(* Logix 5000 project; controller DC01 vendor 1 type 14 code 165 rev 32.12; software revision 32.04; part 6 of 13 *)
(* tags used below, declared in another part *)
   Always_Off : BOOL;
   Barcode_Scan_ln02 : MESSAGE;
   Break_1stStation : BOOL;
   Break_LineWide : BOOL;
   Break_WorkCenter : BOOL;
   Break_Workstation : BOOL;
   FaultExists : CONTROL;
   LN02_MainLine_MSG : MESSAGE;
   Local_Timer : TIMER[30];
   local_timer2 : TIMER;
   ONS_0 : DINT;
   Scheduled_Units_Buffer : DINT;
   Shift_Reset : BOOL;
   Shift_Reset_ONS : BOOL;
   LN02_1st_Station_Break_Code : DINT;
   LN02_Additional_Break_Limit_Mins : DINT;
   LN02_Boxing_MNT : DINT;
   LN02_Ceran_MNT : DINT;
   LN02_Console_MNT : DINT;
   LN02_Cooktop_MNT : DINT;
   LN02_Current_Shift_Duration_Mins : DINT;
   LN02_Current_Shift_Duration_wBreaks_Mins : DINT;
   LN02_DC_Controlled_Theoretical_Units : BOOL;
   LN02_Door_MNT : DINT;
   LN02_FPY : REAL;
   LN02_FrontFrame_MNT : DINT;
   LN02_Ignition_NewSNModel : BOOL[32];
   LN02_Ignition_SNModelMSG : STRING[5];
   LN02_MachineOverAll_MNT : DINT;
   LN02_Main_Messages : DINT[250];
   LN02_MainBack_MNT : DINT;
   LN02_Messages_Barcode_SNModel : Barcode_SNModel;
   LN02_OT_Shift_Break_In_Minutes : DINT;
   LN02_OvenCavity_MNT : DINT;
   LN02_Schedule : UDT_Current_Status;
   LN02_Schedule_Cycle_Timer : TIMER;
   LN02_Schedule_Max_Break_Duration : DINT;
   LN02_Schedule_Max_Break_Timer : TIMER;
   LN02_Schedule_TAKT_REAL : REAL;
   LN02_SidePanels_MNT : DINT;
   LN02_Standard_Shift_Break_In_Minutes : DINT;
   LN02_StorageDrawer_MNT : DINT;
   LN02_Test_MNT : DINT;
   LN02_Theoretical_Units_Counter : COUNTER;
   LN02_Theoretical_Units_Counter_ONS : BOOL;
   LN02_Units_for_repair : DINT;
   LN02_Wiring_MNT : DINT;
   LN02ECM02 : DINT;
   LN02ECM03 : DINT;
   LN02ECM04 : DINT;
   LN02ECM05 : DINT;
   LN02EDM04 : DINT;
   LN02EDM06 : DINT;
   LN02EDM07 : DINT;
   LN02EEM01 : DINT;
   LN02EEM02 : DINT;
   LN02EHM01 : DINT;
   LN02EHM02 : DINT;
   LN02EHM03 : DINT;
   LN02EHM04 : DINT;
   LN02EHM05 : DINT;
   LN02EHM06 : DINT;
   LN02EHM07 : DINT;
   LN02EHM08 : DINT;
   LN02EHM09 : DINT;
   LN02EHM10 : DINT;
   LN02NAS03 : DINT;
   LN02NES01 : DINT;
   LN02NES02 : DINT;
   LN02NES03 : DINT;
   LN02NES04 : DINT;
   LN02NFS01 : DINT;
   LN02NFS02 : DINT;
   LN02SAS01 : DINT;
   LN02SAS02 : DINT;
   LN02SAS03 : DINT;
   LN02SBS01 : DINT;
   LN02SBS02 : DINT;
   LN02SBS03 : DINT;
   LN02SFS01 : DINT;
   LN02SFS02 : DINT;
   LN02SFS03 : DINT;
   LN02SFS04 : DINT;
   LN02WAM01 : DINT;
   LN02WBM01 : DINT;
   LN02WBM02 : DINT;
   LN02WBM03 : DINT;
   LN02WBM04 : DINT;
   LN02WCM01 : DINT;
   LN02WCM02 : DINT;
   LN02WCM03 : DINT;
   LN02WCM04 : DINT;
   LN02WCM05 : DINT;
   LN02WCM06 : DINT;
   LN02WDM01 : DINT;
   LN02WDM02 : DINT;
   LN02WDM03 : DINT;
   LN02WDM04 : DINT;
   LN02WDM05 : DINT;
   LN02WDM06 : DINT;
   LN02WEM01 : DINT;
   LN02WFM01 : DINT;
   LN02WGM01 : DINT;
   LN02WGS01 : DINT;
   LN02WGS02 : DINT;
   LN02WGS03 : DINT;
   LN02WGS04 : DINT;
(* LN02, continued *)

ROUTINE R02_CurrentShift_Calcs   (* ladder *)
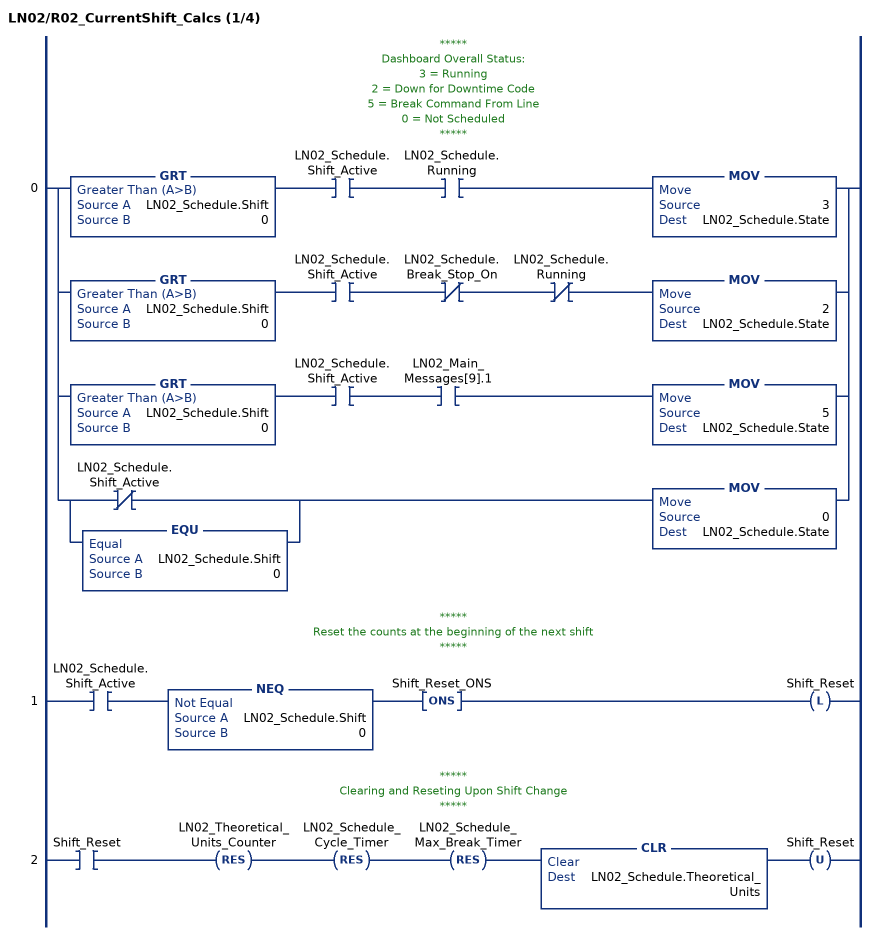
   // *****
   // Dashboard Overall Status:
   // 3 = Running
   // 2 = Down for Downtime Code
   // 5 = Break Command From Line
   // 0 = Not Scheduled
   // *****
   0: [GRT(LN02_Schedule.Shift,0) XIC(LN02_Schedule.Shift_Active) XIC(LN02_Schedule.Running) MOV(3,LN02_Schedule.State) ,GRT(LN02_Schedule.Shift,0) XIC(LN02_Schedule.Shift_Active) XIO(LN02_Schedule.Break_Stop_On) XIO(LN02_Schedule.Running) MOV(2,LN02_Schedule.State) ,GRT(LN02_Schedule.Shift,0) XIC(LN02_Schedule.Shift_Active) XIC(LN02_Main_Messages[9].1) MOV(5,LN02_Schedule.State) ,[XIO(LN02_Schedule.Shift_Active) ,EQU(LN02_Schedule.Shift,0) ] MOV(0,LN02_Schedule.State) ];
   // *****
   // Reset the counts at the beginning of the next shift
   // *****
   1: XIC(LN02_Schedule.Shift_Active)NEQ(LN02_Schedule.Shift,0)ONS(Shift_Reset_ONS)OTL(Shift_Reset);
   // *****
   // Clearing and Reseting Upon Shift Change
   // *****
   2: XIC(Shift_Reset)RES(LN02_Theoretical_Units_Counter)RES(LN02_Schedule_Cycle_Timer)RES(LN02_Schedule_Max_Break_Timer)CLR(LN02_Schedule.Theoretical_Units)OTU(Shift_Reset);
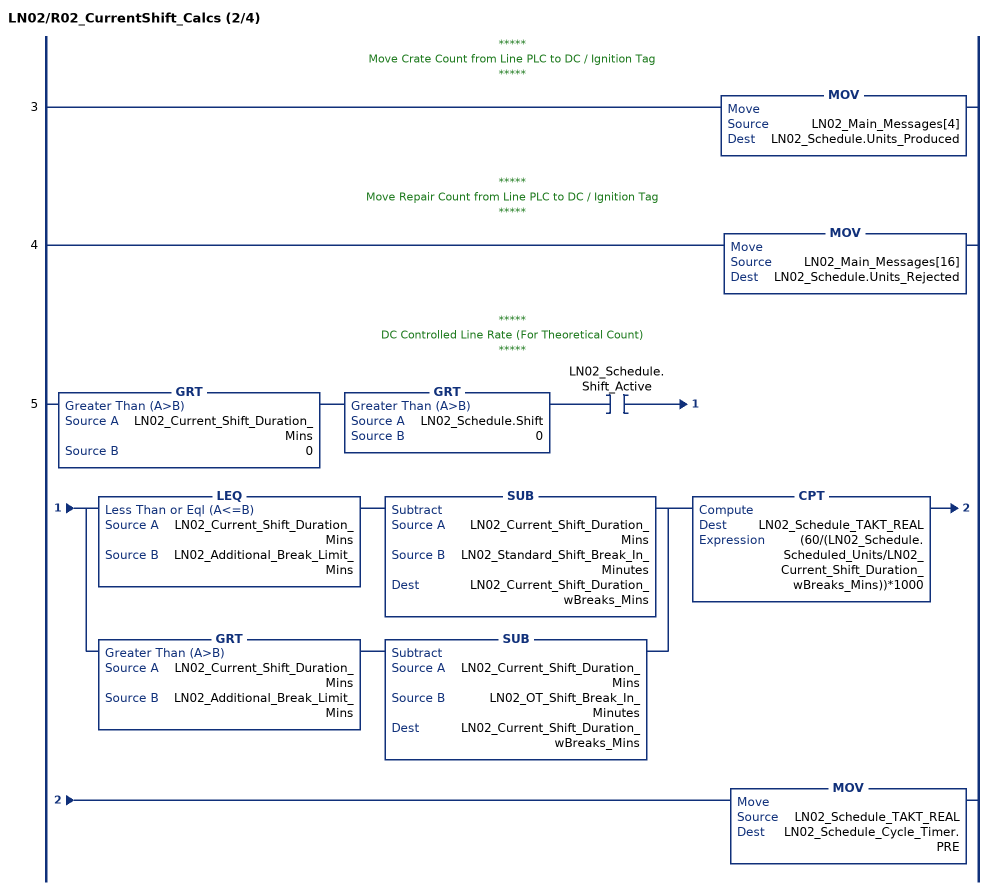
   // *****
   // Move Crate Count from Line PLC to DC / Ignition Tag
   // *****
   3: MOV(LN02_Main_Messages[4],LN02_Schedule.Units_Produced);
   // *****
   // Move Repair Count from Line PLC to DC / Ignition Tag
   // *****
   4: MOV(LN02_Main_Messages[16],LN02_Schedule.Units_Rejected);
   // *****
   // DC Controlled Line Rate (For Theoretical Count)
   // *****
   5: GRT(LN02_Current_Shift_Duration_Mins,0)GRT(LN02_Schedule.Shift,0)XIC(LN02_Schedule.Shift_Active)[LEQ(LN02_Current_Shift_Duration_Mins,LN02_Additional_Break_Limit_Mins) SUB(LN02_Current_Shift_Duration_Mins,LN02_Standard_Shift_Break_In_Minutes,LN02_Current_Shift_Duration_wBreaks_Mins) ,GRT(LN02_Current_Shift_Duration_Mins,LN02_Additional_Break_Limit_Mins) SUB(LN02_Current_Shift_Duration_Mins,LN02_OT_Shift_Break_In_Minutes,LN02_Current_Shift_Duration_wBreaks_Mins) ]CPT(LN02_Schedule_TAKT_REAL,(60/(LN02_Schedule.Scheduled_Units/LN02_Current_Shift_Duration_wBreaks_Mins))*1000)MOV(LN02_Schedule_TAKT_REAL,LN02_Schedule_Cycle_Timer.PRE);
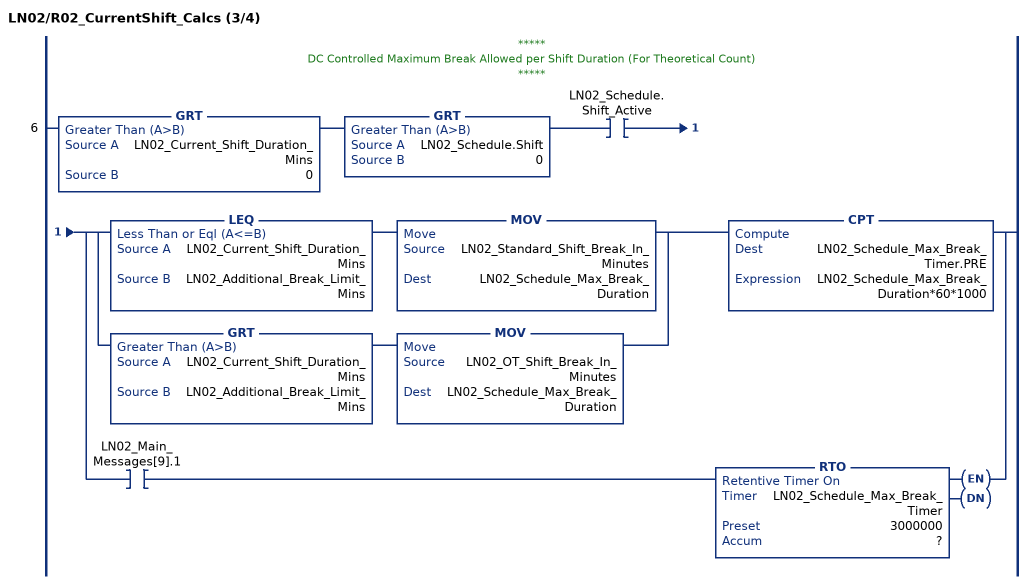
   // *****
   // DC Controlled Maximum Break Allowed per Shift Duration (For Theoretical Count)
   // *****
   6: GRT(LN02_Current_Shift_Duration_Mins,0)GRT(LN02_Schedule.Shift,0)XIC(LN02_Schedule.Shift_Active)[[LEQ(LN02_Current_Shift_Duration_Mins,LN02_Additional_Break_Limit_Mins) MOV(LN02_Standard_Shift_Break_In_Minutes,LN02_Schedule_Max_Break_Duration) ,GRT(LN02_Current_Shift_Duration_Mins,LN02_Additional_Break_Limit_Mins) MOV(LN02_OT_Shift_Break_In_Minutes,LN02_Schedule_Max_Break_Duration) ] CPT(LN02_Schedule_Max_Break_Timer.PRE,LN02_Schedule_Max_Break_Duration*60*1000) ,XIC(LN02_Main_Messages[9].1) RTO(LN02_Schedule_Max_Break_Timer,?,?) ];
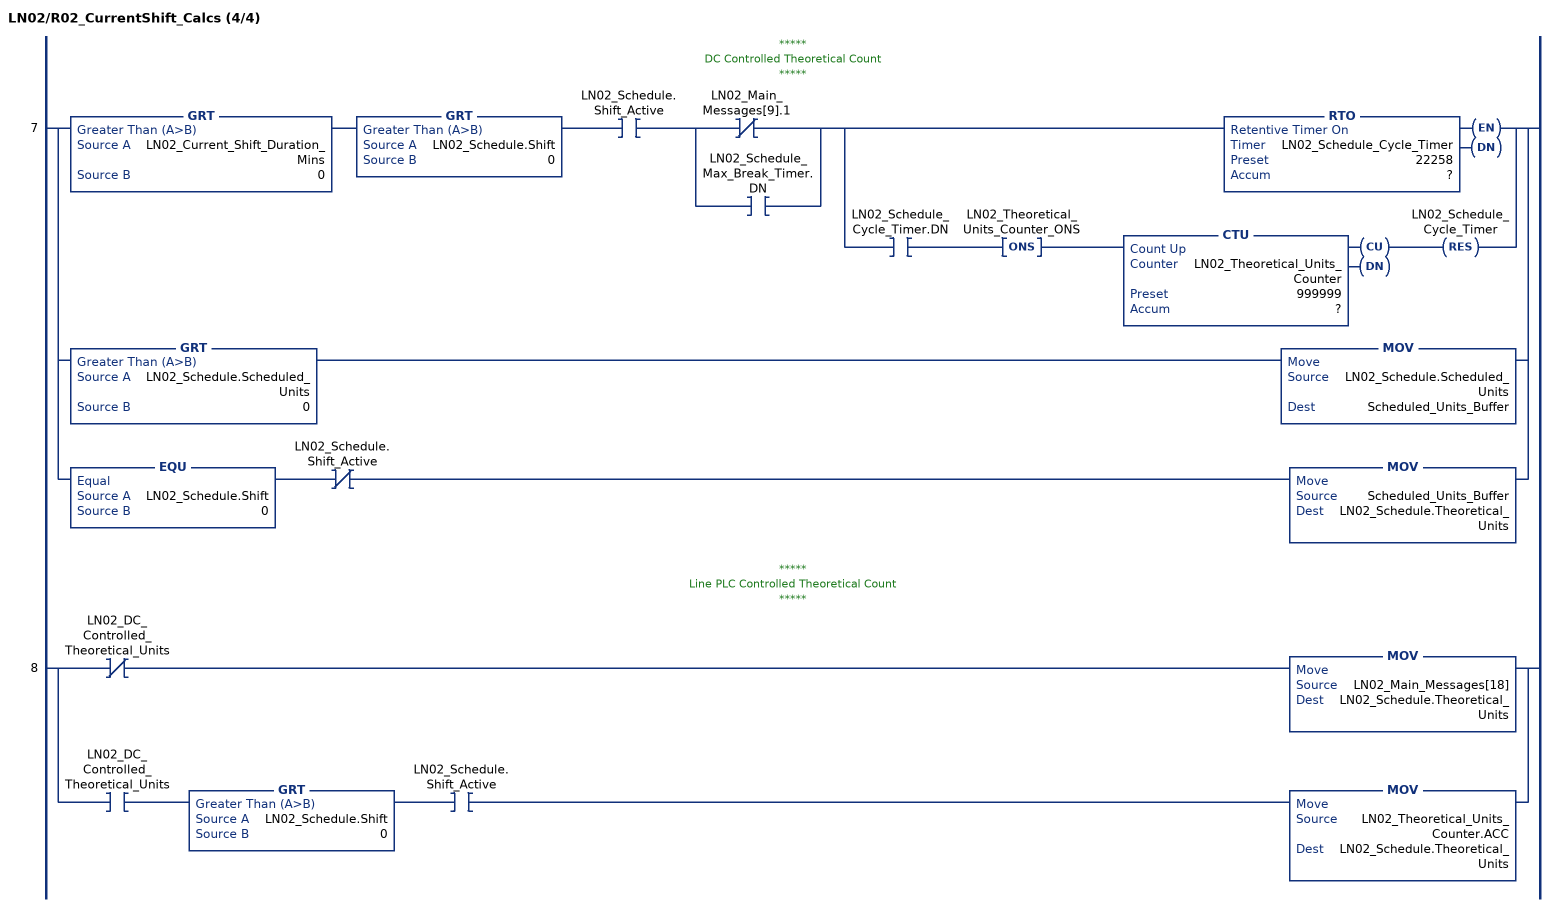
   // *****
   // DC Controlled Theoretical Count
   // *****
   7: [GRT(LN02_Current_Shift_Duration_Mins,0) GRT(LN02_Schedule.Shift,0) XIC(LN02_Schedule.Shift_Active) [XIO(LN02_Main_Messages[9].1) ,XIC(LN02_Schedule_Max_Break_Timer.DN) ] [RTO(LN02_Schedule_Cycle_Timer,?,?) ,XIC(LN02_Schedule_Cycle_Timer.DN) ONS(LN02_Theoretical_Units_Counter_ONS) CTU(LN02_Theoretical_Units_Counter,?,?) RES(LN02_Schedule_Cycle_Timer) ] ,GRT(LN02_Schedule.Scheduled_Units,0) MOV(LN02_Schedule.Scheduled_Units,Scheduled_Units_Buffer) ,EQU(LN02_Schedule.Shift,0) XIO(LN02_Schedule.Shift_Active) MOV(Scheduled_Units_Buffer,LN02_Schedule.Theoretical_Units) ];
   // *****
   // Line PLC Controlled Theoretical Count
   // *****
   8: [XIO(LN02_DC_Controlled_Theoretical_Units) MOV(LN02_Main_Messages[18],LN02_Schedule.Theoretical_Units) ,XIC(LN02_DC_Controlled_Theoretical_Units) GRT(LN02_Schedule.Shift,0) XIC(LN02_Schedule.Shift_Active) MOV(LN02_Theoretical_Units_Counter.ACC,LN02_Schedule.Theoretical_Units) ];
END_ROUTINE

ROUTINE R03_DataFromLines   (* ladder *)
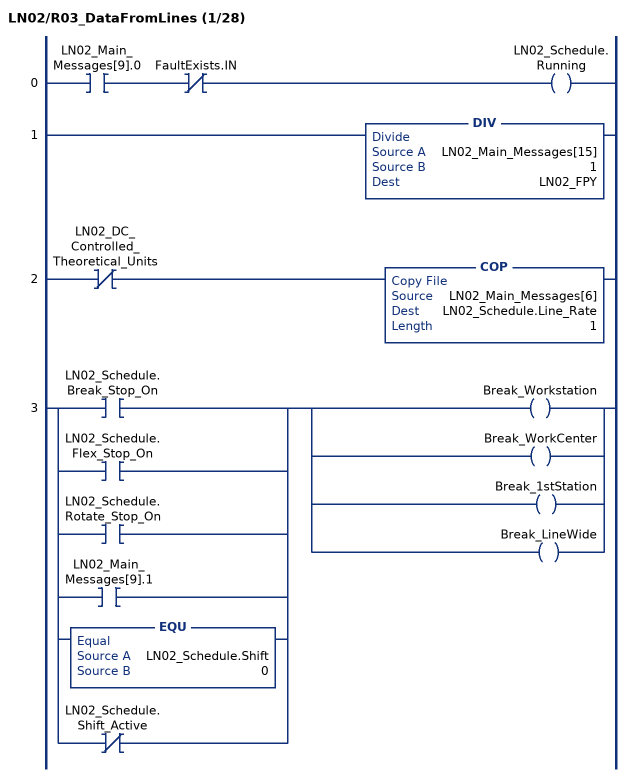
   0: XIC(LN02_Main_Messages[9].0)XIO(FaultExists.IN)OTE(LN02_Schedule.Running);
   1: DIV(LN02_Main_Messages[15],1,LN02_FPY);
   2: XIO(LN02_DC_Controlled_Theoretical_Units)COP(LN02_Main_Messages[6],LN02_Schedule.Line_Rate,1);
   3: [XIC(LN02_Schedule.Break_Stop_On) ,XIC(LN02_Schedule.Flex_Stop_On) ,XIC(LN02_Schedule.Rotate_Stop_On) ,XIC(LN02_Main_Messages[9].1) ,EQU(LN02_Schedule.Shift,0) ,XIO(LN02_Schedule.Shift_Active) ][OTE(Break_Workstation) ,OTE(Break_WorkCenter) ,OTE(Break_1stStation) ,OTE(Break_LineWide) ];
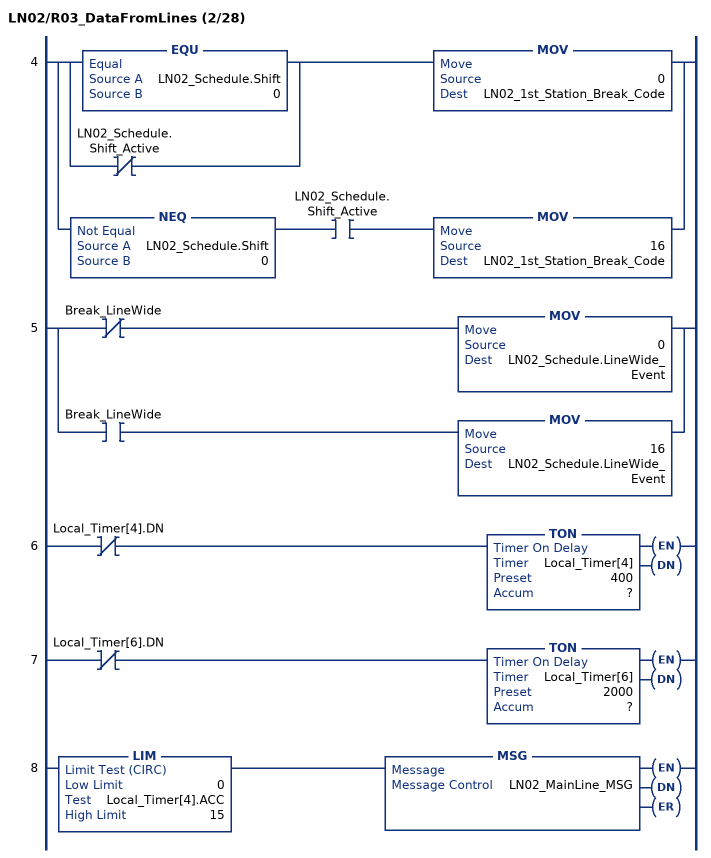
   4: [[EQU(LN02_Schedule.Shift,0) ,XIO(LN02_Schedule.Shift_Active) ] MOV(0,LN02_1st_Station_Break_Code) ,NEQ(LN02_Schedule.Shift,0) XIC(LN02_Schedule.Shift_Active) MOV(16,LN02_1st_Station_Break_Code) ];
   5: [XIO(Break_LineWide) MOV(0,LN02_Schedule.LineWide_Event) ,XIC(Break_LineWide) MOV(16,LN02_Schedule.LineWide_Event) ];
   6: XIO(Local_Timer[4].DN)TON(Local_Timer[4],?,?);
   7: XIO(Local_Timer[6].DN)TON(Local_Timer[6],?,?);
   8: LIM(0,Local_Timer[4].ACC,15)MSG(LN02_MainLine_MSG);
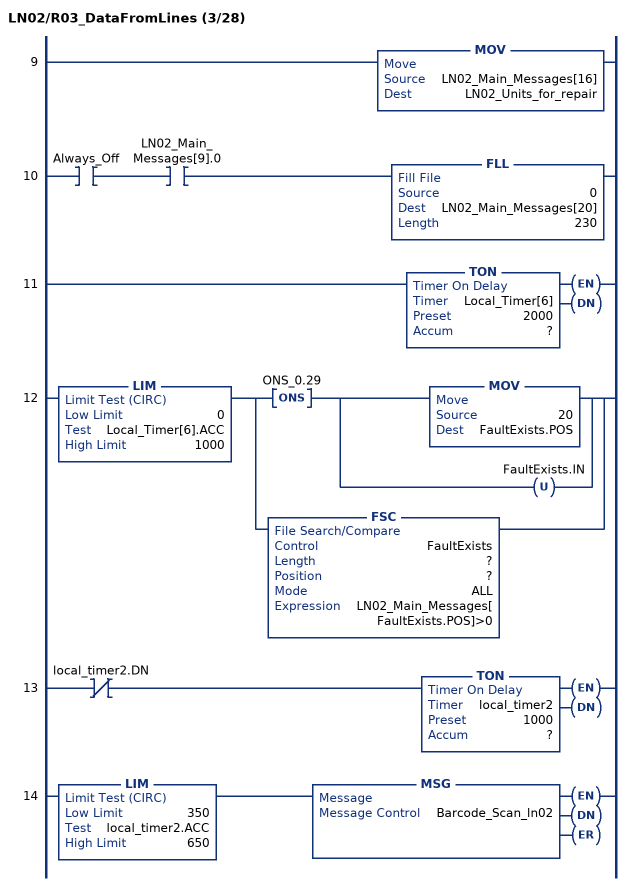
   9: MOV(LN02_Main_Messages[16],LN02_Units_for_repair);
   10: XIC(Always_Off)XIC(LN02_Main_Messages[9].0)FLL(0,LN02_Main_Messages[20],230);
   11: TON(Local_Timer[6],?,?);
   12: LIM(0,Local_Timer[6].ACC,1000)[ONS(ONS_0.29) [MOV(20,FaultExists.POS) ,OTU(FaultExists.IN) ] ,FSC(FaultExists,?,?,ALL,LN02_Main_Messages[FaultExists.POS]>0) ];
   13: XIO(local_timer2.DN)TON(local_timer2,?,?);
   14: LIM(350,local_timer2.ACC,650)MSG(Barcode_Scan_ln02);
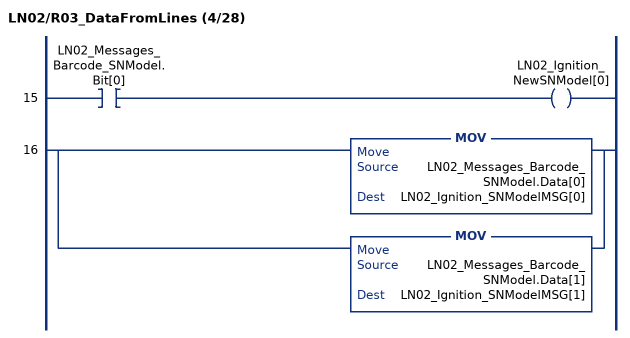
   15: XIC(LN02_Messages_Barcode_SNModel.Bit[0])OTE(LN02_Ignition_NewSNModel[0]);
   16: [MOV(LN02_Messages_Barcode_SNModel.Data[0],LN02_Ignition_SNModelMSG[0]) ,MOV(LN02_Messages_Barcode_SNModel.Data[1],LN02_Ignition_SNModelMSG[1]) ];
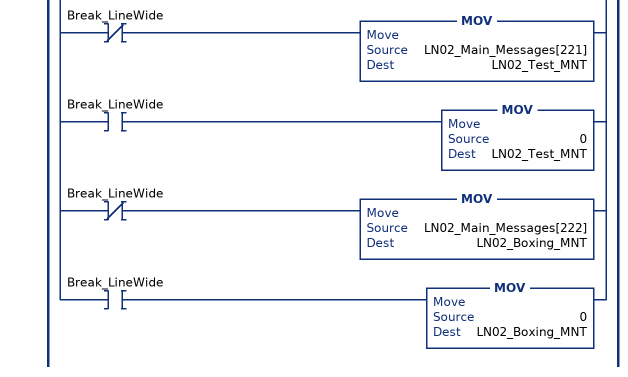
   // MNT Faults
   // If an MNT workcenter is tied to the main line or subline where there is already a workcenter with a workstaiton where "Break_LineWide (when high) MOVEs a 16 in, then that MNT can MOVE a 0 in when "Break_LineWide" goes high
   // If it is an independent MNT (not tied to a workcenter), "Break_LineWide" Tag should MOVE a 16 when "Break_LineWide" goes high
   17: [XIO(Break_LineWide) MOV(LN02_Main_Messages[20],LN02_MachineOverAll_MNT) ,XIC(Break_LineWide) MOV(0,LN02_MachineOverAll_MNT) ,XIO(Break_LineWide) MOV(LN02_Main_Messages[21],LN02_FrontFrame_MNT) ,XIC(Break_LineWide) MOV(0,LN02_FrontFrame_MNT) ,XIO(Break_LineWide) MOV(LN02_Main_Messages[22],LN02_OvenCavity_MNT) ,XIC(Break_LineWide) MOV(0,LN02_OvenCavity_MNT) ,XIO(Break_LineWide) MOV(LN02_Main_Messages[23],LN02_MainBack_MNT) ,XIC(Break_LineWide) MOV(0,LN02_MainBack_MNT) ,XIO(Break_LineWide) MOV(LN02_Main_Messages[24],LN02_SidePanels_MNT) ,XIC(Break_LineWide) MOV(0,LN02_SidePanels_MNT) ,XIO(Break_LineWide) MOV(LN02_Main_Messages[25],LN02_Console_MNT) ,XIC(Break_LineWide) MOV(0,LN02_Console_MNT) ,XIO(Break_LineWide) MOV(LN02_Main_Messages[26],LN02_Cooktop_MNT) ,XIC(Break_LineWide) MOV(0,LN02_Cooktop_MNT) ,XIO(Break_LineWide) MOV(LN02_Main_Messages[27],LN02_Ceran_MNT) ,XIC(Break_LineWide) MOV(0,LN02_Ceran_MNT) ,XIO(Break_LineWide) MOV(LN02_Main_Messages[28],LN02_Wiring_MNT) ,XIC(Break_LineWide) MOV(0,LN02_Wiring_MNT) ,XIO(Break_LineWide) MOV(LN02_Main_Messages[29],LN02_StorageDrawer_MNT) ,XIC(Break_LineWide) MOV(0,LN02_StorageDrawer_MNT) ,XIO(Break_LineWide) MOV(LN02_Main_Messages[220],LN02_Door_MNT) ,XIC(Break_LineWide) MOV(0,LN02_Door_MNT) ,XIO(Break_LineWide) MOV(LN02_Main_Messages[221],LN02_Test_MNT) ,XIC(Break_LineWide) MOV(0,LN02_Test_MNT) ,XIO(Break_LineWide) MOV(LN02_Main_Messages[222],LN02_Boxing_MNT) ,XIC(Break_LineWide) MOV(0,LN02_Boxing_MNT) ];
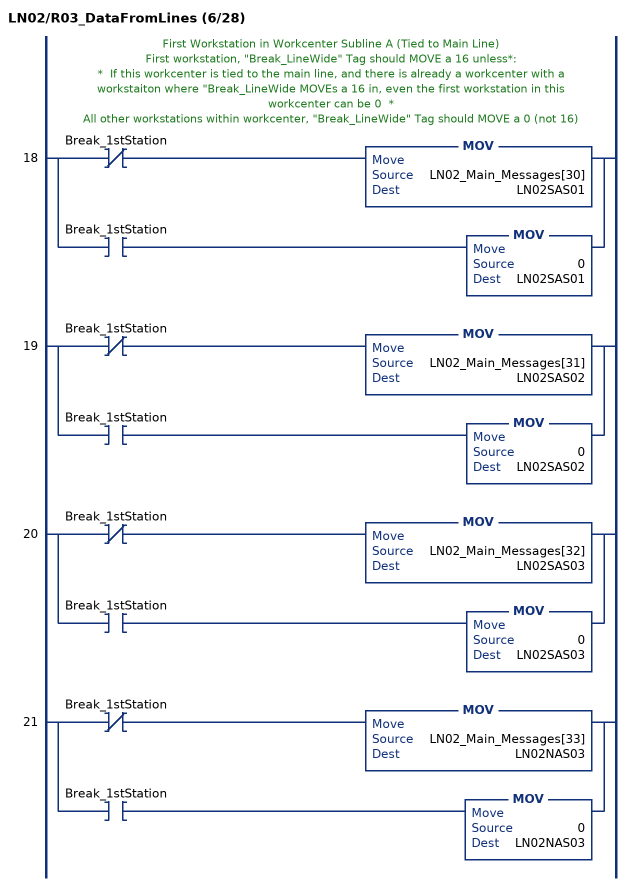
   // First Workstation in Workcenter Subline A (Tied to Main Line)
   // First workstation, "Break_LineWide" Tag should MOVE a 16 unless*:
   // *  If this workcenter is tied to the main line, and there is already a workcenter with a workstaiton where "Break_LineWide MOVEs a 16 in, even the first workstation in this workcenter can be 0  *
   // All other workstations within workcenter, "Break_LineWide" Tag should MOVE a 0 (not 16)
   18: [XIO(Break_1stStation) MOV(LN02_Main_Messages[30],LN02SAS01) ,XIC(Break_1stStation) MOV(0,LN02SAS01) ];
   19: [XIO(Break_1stStation) MOV(LN02_Main_Messages[31],LN02SAS02) ,XIC(Break_1stStation) MOV(0,LN02SAS02) ];
   20: [XIO(Break_1stStation) MOV(LN02_Main_Messages[32],LN02SAS03) ,XIC(Break_1stStation) MOV(0,LN02SAS03) ];
   21: [XIO(Break_1stStation) MOV(LN02_Main_Messages[33],LN02NAS03) ,XIC(Break_1stStation) MOV(0,LN02NAS03) ];
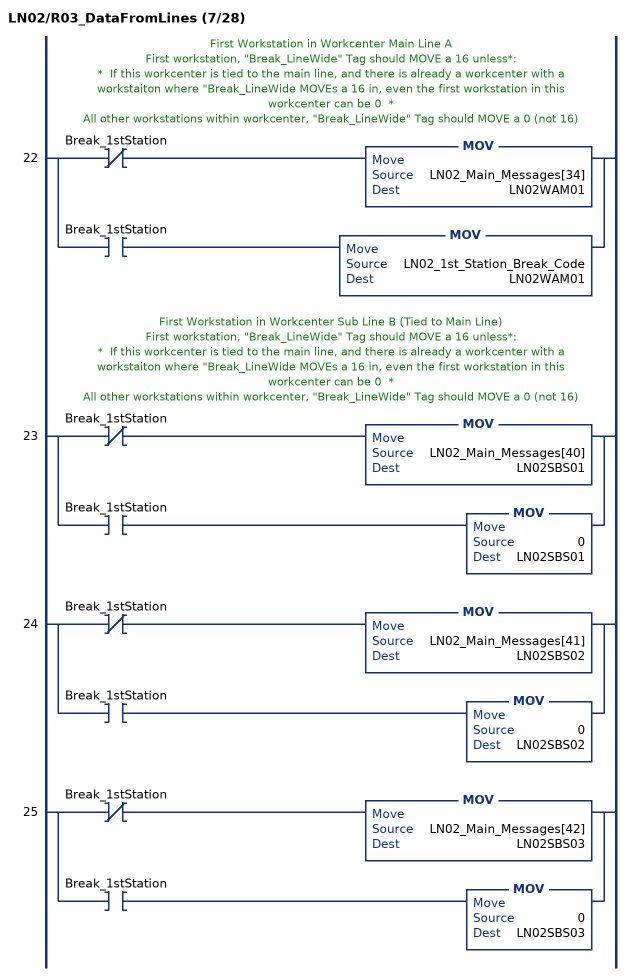
   // First Workstation in Workcenter Main Line A
   // First workstation, "Break_LineWide" Tag should MOVE a 16 unless*:
   // *  If this workcenter is tied to the main line, and there is already a workcenter with a workstaiton where "Break_LineWide MOVEs a 16 in, even the first workstation in this workcenter can be 0  *
   // All other workstations within workcenter, "Break_LineWide" Tag should MOVE a 0 (not 16)
   22: [XIO(Break_1stStation) MOV(LN02_Main_Messages[34],LN02WAM01) ,XIC(Break_1stStation) MOV(LN02_1st_Station_Break_Code,LN02WAM01) ];
   // First Workstation in Workcenter Sub Line B (Tied to Main Line)
   // First workstation, "Break_LineWide" Tag should MOVE a 16 unless*:
   // *  If this workcenter is tied to the main line, and there is already a workcenter with a workstaiton where "Break_LineWide MOVEs a 16 in, even the first workstation in this workcenter can be 0  *
   // All other workstations within workcenter, "Break_LineWide" Tag should MOVE a 0 (not 16)
   23: [XIO(Break_1stStation) MOV(LN02_Main_Messages[40],LN02SBS01) ,XIC(Break_1stStation) MOV(0,LN02SBS01) ];
   24: [XIO(Break_1stStation) MOV(LN02_Main_Messages[41],LN02SBS02) ,XIC(Break_1stStation) MOV(0,LN02SBS02) ];
   25: [XIO(Break_1stStation) MOV(LN02_Main_Messages[42],LN02SBS03) ,XIC(Break_1stStation) MOV(0,LN02SBS03) ];
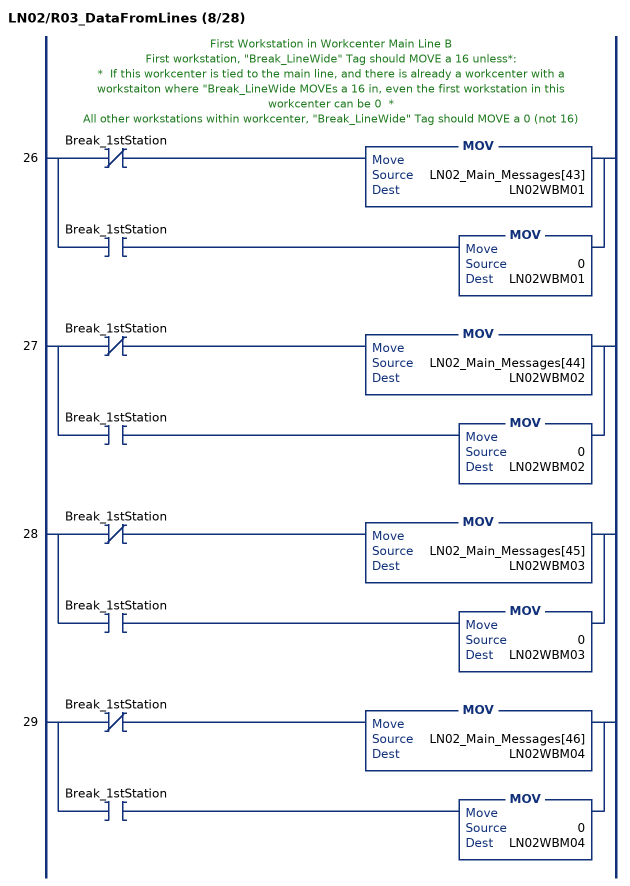
   // First Workstation in Workcenter Main Line B
   // First workstation, "Break_LineWide" Tag should MOVE a 16 unless*:
   // *  If this workcenter is tied to the main line, and there is already a workcenter with a workstaiton where "Break_LineWide MOVEs a 16 in, even the first workstation in this workcenter can be 0  *
   // All other workstations within workcenter, "Break_LineWide" Tag should MOVE a 0 (not 16)
   26: [XIO(Break_1stStation) MOV(LN02_Main_Messages[43],LN02WBM01) ,XIC(Break_1stStation) MOV(0,LN02WBM01) ];
   27: [XIO(Break_1stStation) MOV(LN02_Main_Messages[44],LN02WBM02) ,XIC(Break_1stStation) MOV(0,LN02WBM02) ];
   28: [XIO(Break_1stStation) MOV(LN02_Main_Messages[45],LN02WBM03) ,XIC(Break_1stStation) MOV(0,LN02WBM03) ];
   29: [XIO(Break_1stStation) MOV(LN02_Main_Messages[46],LN02WBM04) ,XIC(Break_1stStation) MOV(0,LN02WBM04) ];
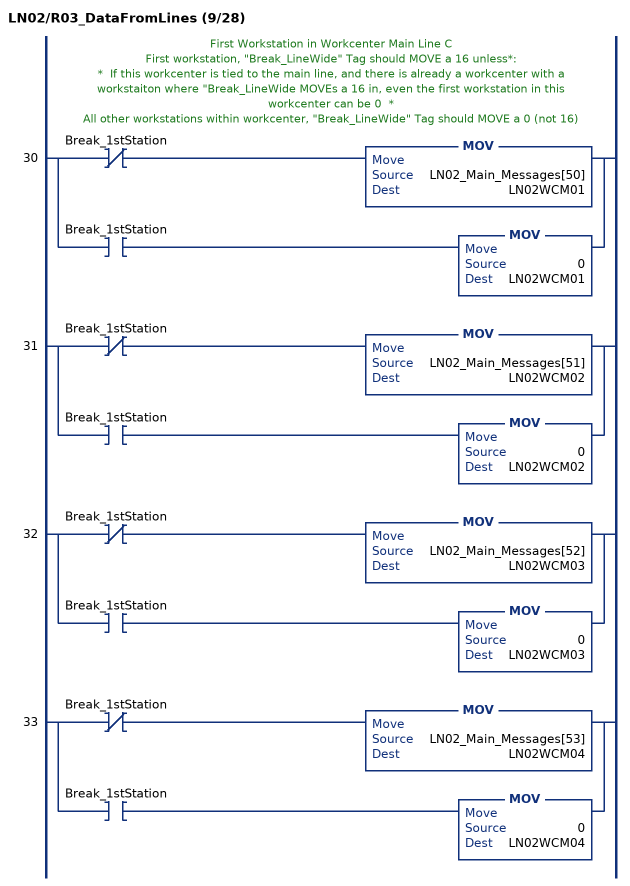
   // First Workstation in Workcenter Main Line C
   // First workstation, "Break_LineWide" Tag should MOVE a 16 unless*:
   // *  If this workcenter is tied to the main line, and there is already a workcenter with a workstaiton where "Break_LineWide MOVEs a 16 in, even the first workstation in this workcenter can be 0  *
   // All other workstations within workcenter, "Break_LineWide" Tag should MOVE a 0 (not 16)
   30: [XIO(Break_1stStation) MOV(LN02_Main_Messages[50],LN02WCM01) ,XIC(Break_1stStation) MOV(0,LN02WCM01) ];
   31: [XIO(Break_1stStation) MOV(LN02_Main_Messages[51],LN02WCM02) ,XIC(Break_1stStation) MOV(0,LN02WCM02) ];
   32: [XIO(Break_1stStation) MOV(LN02_Main_Messages[52],LN02WCM03) ,XIC(Break_1stStation) MOV(0,LN02WCM03) ];
   33: [XIO(Break_1stStation) MOV(LN02_Main_Messages[53],LN02WCM04) ,XIC(Break_1stStation) MOV(0,LN02WCM04) ];
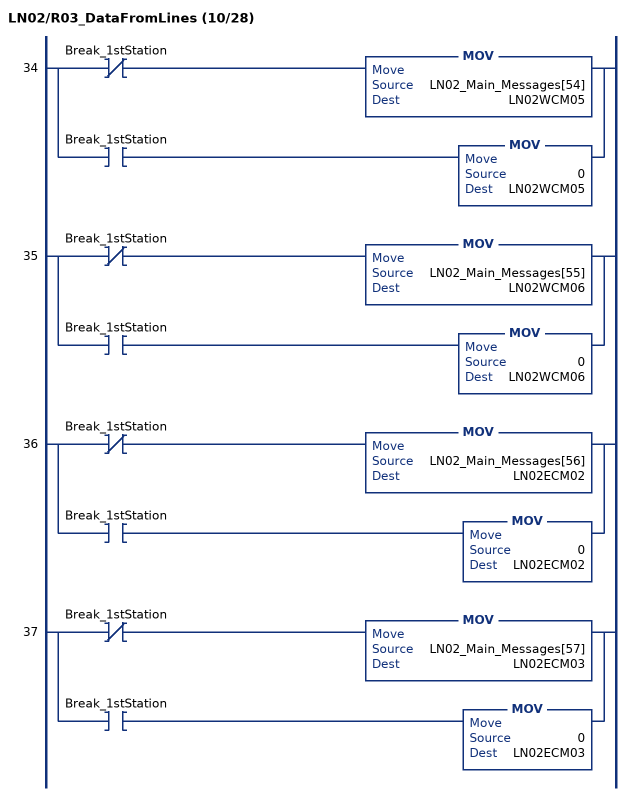
   34: [XIO(Break_1stStation) MOV(LN02_Main_Messages[54],LN02WCM05) ,XIC(Break_1stStation) MOV(0,LN02WCM05) ];
   35: [XIO(Break_1stStation) MOV(LN02_Main_Messages[55],LN02WCM06) ,XIC(Break_1stStation) MOV(0,LN02WCM06) ];
   36: [XIO(Break_1stStation) MOV(LN02_Main_Messages[56],LN02ECM02) ,XIC(Break_1stStation) MOV(0,LN02ECM02) ];
   37: [XIO(Break_1stStation) MOV(LN02_Main_Messages[57],LN02ECM03) ,XIC(Break_1stStation) MOV(0,LN02ECM03) ];
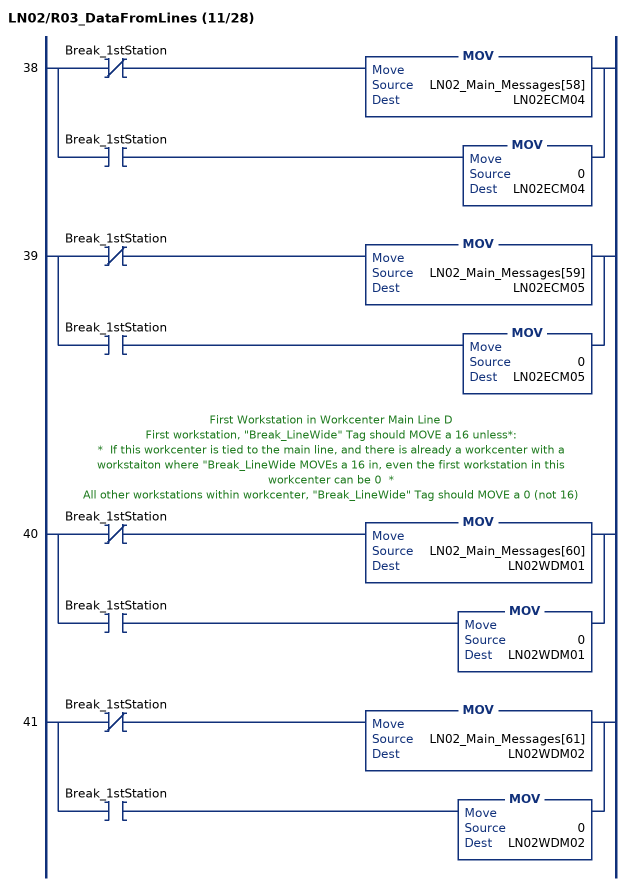
   38: [XIO(Break_1stStation) MOV(LN02_Main_Messages[58],LN02ECM04) ,XIC(Break_1stStation) MOV(0,LN02ECM04) ];
   39: [XIO(Break_1stStation) MOV(LN02_Main_Messages[59],LN02ECM05) ,XIC(Break_1stStation) MOV(0,LN02ECM05) ];
   // First Workstation in Workcenter Main Line D
   // First workstation, "Break_LineWide" Tag should MOVE a 16 unless*:
   // *  If this workcenter is tied to the main line, and there is already a workcenter with a workstaiton where "Break_LineWide MOVEs a 16 in, even the first workstation in this workcenter can be 0  *
   // All other workstations within workcenter, "Break_LineWide" Tag should MOVE a 0 (not 16)
   40: [XIO(Break_1stStation) MOV(LN02_Main_Messages[60],LN02WDM01) ,XIC(Break_1stStation) MOV(0,LN02WDM01) ];
   41: [XIO(Break_1stStation) MOV(LN02_Main_Messages[61],LN02WDM02) ,XIC(Break_1stStation) MOV(0,LN02WDM02) ];
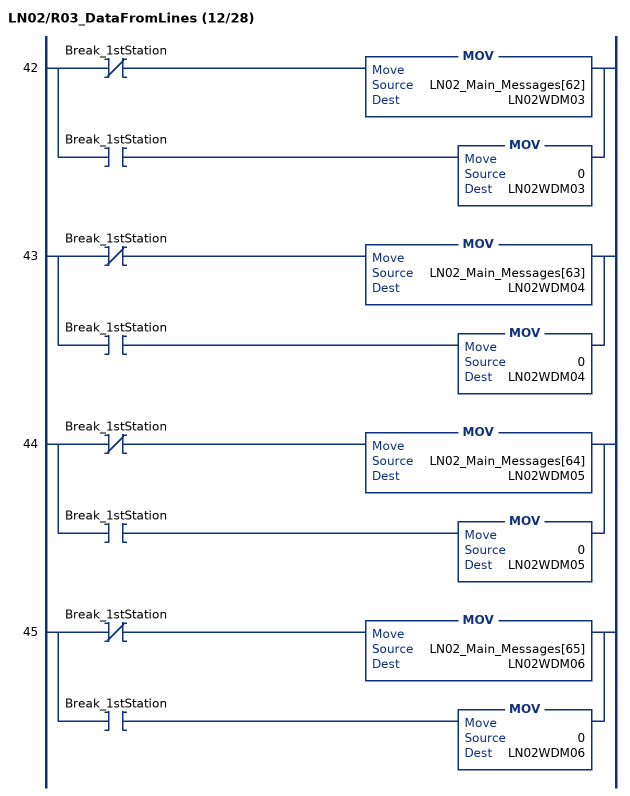
   42: [XIO(Break_1stStation) MOV(LN02_Main_Messages[62],LN02WDM03) ,XIC(Break_1stStation) MOV(0,LN02WDM03) ];
   43: [XIO(Break_1stStation) MOV(LN02_Main_Messages[63],LN02WDM04) ,XIC(Break_1stStation) MOV(0,LN02WDM04) ];
   44: [XIO(Break_1stStation) MOV(LN02_Main_Messages[64],LN02WDM05) ,XIC(Break_1stStation) MOV(0,LN02WDM05) ];
   45: [XIO(Break_1stStation) MOV(LN02_Main_Messages[65],LN02WDM06) ,XIC(Break_1stStation) MOV(0,LN02WDM06) ];
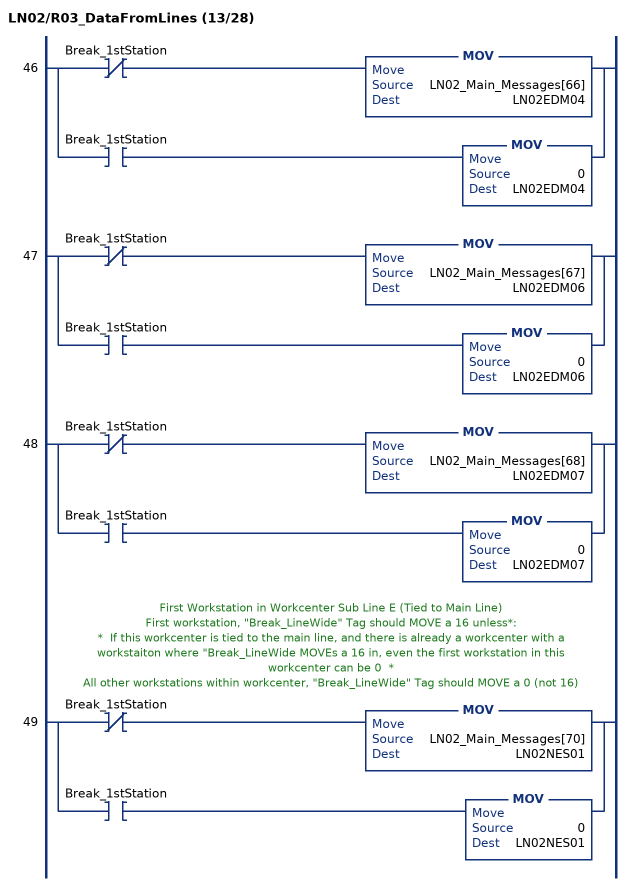
   46: [XIO(Break_1stStation) MOV(LN02_Main_Messages[66],LN02EDM04) ,XIC(Break_1stStation) MOV(0,LN02EDM04) ];
   47: [XIO(Break_1stStation) MOV(LN02_Main_Messages[67],LN02EDM06) ,XIC(Break_1stStation) MOV(0,LN02EDM06) ];
   48: [XIO(Break_1stStation) MOV(LN02_Main_Messages[68],LN02EDM07) ,XIC(Break_1stStation) MOV(0,LN02EDM07) ];
   // First Workstation in Workcenter Sub Line E (Tied to Main Line)
   // First workstation, "Break_LineWide" Tag should MOVE a 16 unless*:
   // *  If this workcenter is tied to the main line, and there is already a workcenter with a workstaiton where "Break_LineWide MOVEs a 16 in, even the first workstation in this workcenter can be 0  *
   // All other workstations within workcenter, "Break_LineWide" Tag should MOVE a 0 (not 16)
   49: [XIO(Break_1stStation) MOV(LN02_Main_Messages[70],LN02NES01) ,XIC(Break_1stStation) MOV(0,LN02NES01) ];
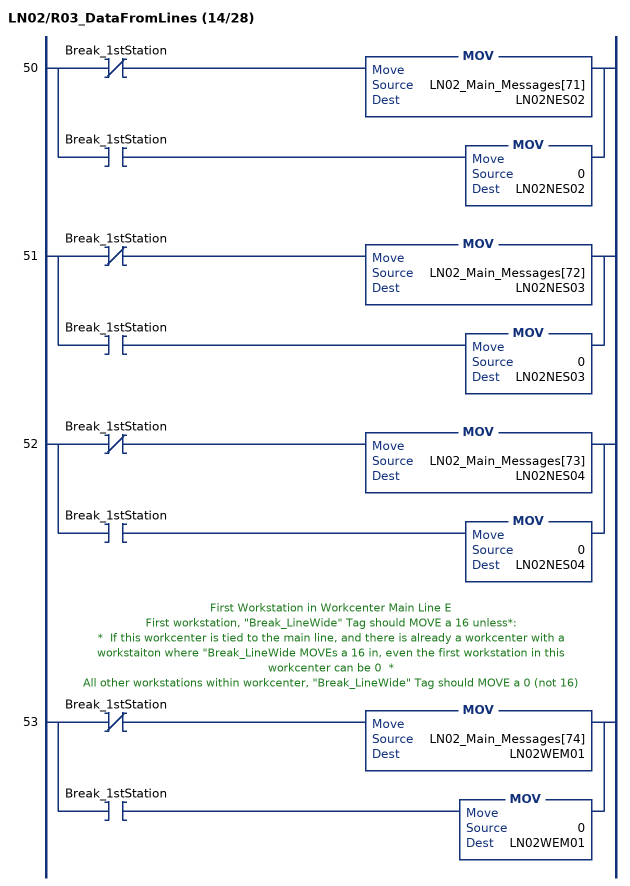
   50: [XIO(Break_1stStation) MOV(LN02_Main_Messages[71],LN02NES02) ,XIC(Break_1stStation) MOV(0,LN02NES02) ];
   51: [XIO(Break_1stStation) MOV(LN02_Main_Messages[72],LN02NES03) ,XIC(Break_1stStation) MOV(0,LN02NES03) ];
   52: [XIO(Break_1stStation) MOV(LN02_Main_Messages[73],LN02NES04) ,XIC(Break_1stStation) MOV(0,LN02NES04) ];
   // First Workstation in Workcenter Main Line E
   // First workstation, "Break_LineWide" Tag should MOVE a 16 unless*:
   // *  If this workcenter is tied to the main line, and there is already a workcenter with a workstaiton where "Break_LineWide MOVEs a 16 in, even the first workstation in this workcenter can be 0  *
   // All other workstations within workcenter, "Break_LineWide" Tag should MOVE a 0 (not 16)
   53: [XIO(Break_1stStation) MOV(LN02_Main_Messages[74],LN02WEM01) ,XIC(Break_1stStation) MOV(0,LN02WEM01) ];
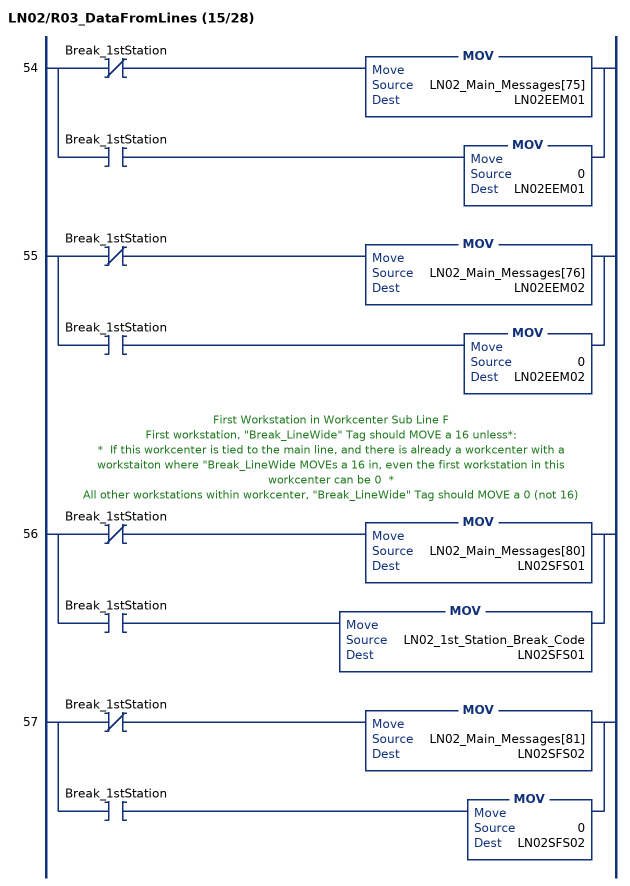
   54: [XIO(Break_1stStation) MOV(LN02_Main_Messages[75],LN02EEM01) ,XIC(Break_1stStation) MOV(0,LN02EEM01) ];
   55: [XIO(Break_1stStation) MOV(LN02_Main_Messages[76],LN02EEM02) ,XIC(Break_1stStation) MOV(0,LN02EEM02) ];
   // First Workstation in Workcenter Sub Line F
   // First workstation, "Break_LineWide" Tag should MOVE a 16 unless*:
   // *  If this workcenter is tied to the main line, and there is already a workcenter with a workstaiton where "Break_LineWide MOVEs a 16 in, even the first workstation in this workcenter can be 0  *
   // All other workstations within workcenter, "Break_LineWide" Tag should MOVE a 0 (not 16)
   56: [XIO(Break_1stStation) MOV(LN02_Main_Messages[80],LN02SFS01) ,XIC(Break_1stStation) MOV(LN02_1st_Station_Break_Code,LN02SFS01) ];
   57: [XIO(Break_1stStation) MOV(LN02_Main_Messages[81],LN02SFS02) ,XIC(Break_1stStation) MOV(0,LN02SFS02) ];
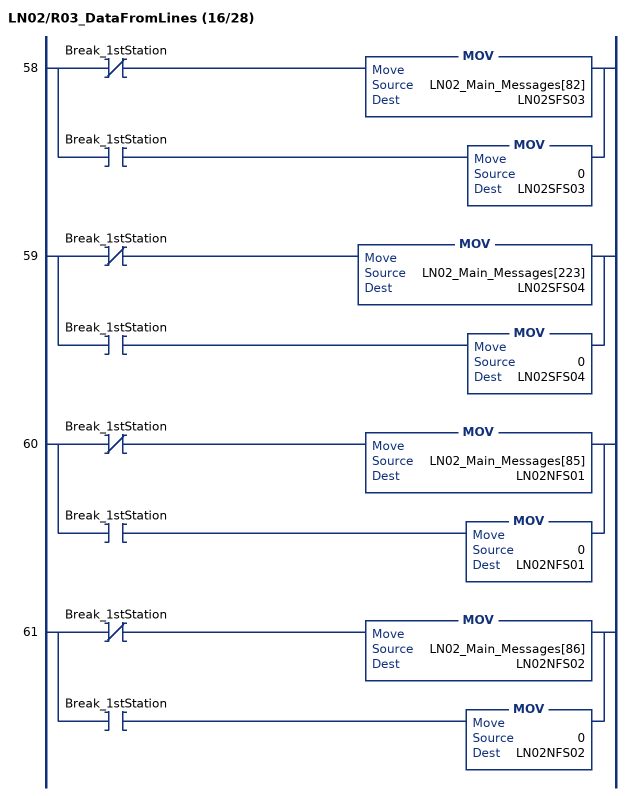
   58: [XIO(Break_1stStation) MOV(LN02_Main_Messages[82],LN02SFS03) ,XIC(Break_1stStation) MOV(0,LN02SFS03) ];
   59: [XIO(Break_1stStation) MOV(LN02_Main_Messages[223],LN02SFS04) ,XIC(Break_1stStation) MOV(0,LN02SFS04) ];
   60: [XIO(Break_1stStation) MOV(LN02_Main_Messages[85],LN02NFS01) ,XIC(Break_1stStation) MOV(0,LN02NFS01) ];
   61: [XIO(Break_1stStation) MOV(LN02_Main_Messages[86],LN02NFS02) ,XIC(Break_1stStation) MOV(0,LN02NFS02) ];
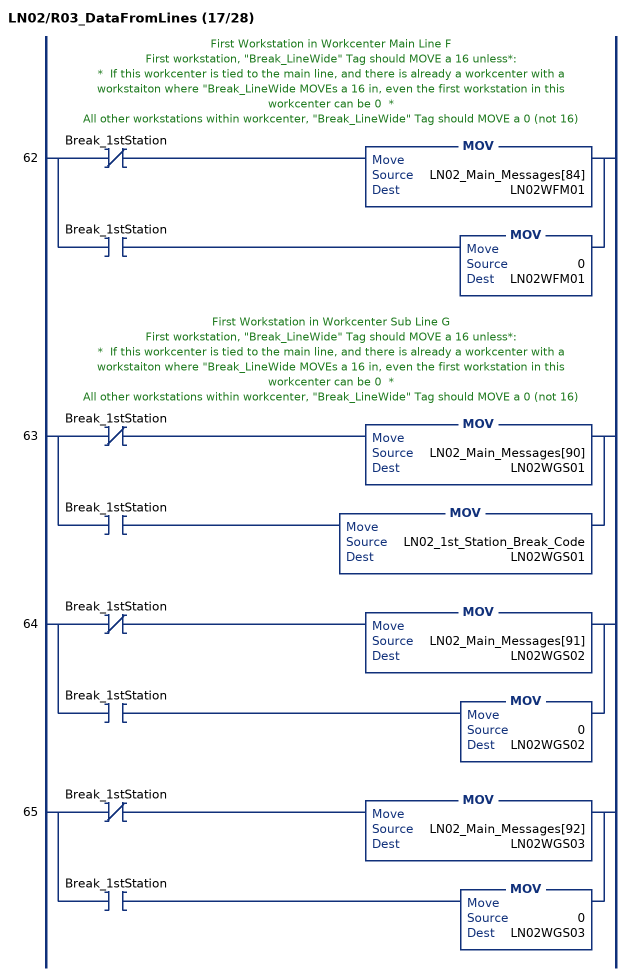
   // First Workstation in Workcenter Main Line F
   // First workstation, "Break_LineWide" Tag should MOVE a 16 unless*:
   // *  If this workcenter is tied to the main line, and there is already a workcenter with a workstaiton where "Break_LineWide MOVEs a 16 in, even the first workstation in this workcenter can be 0  *
   // All other workstations within workcenter, "Break_LineWide" Tag should MOVE a 0 (not 16)
   62: [XIO(Break_1stStation) MOV(LN02_Main_Messages[84],LN02WFM01) ,XIC(Break_1stStation) MOV(0,LN02WFM01) ];
   // First Workstation in Workcenter Sub Line G
   // First workstation, "Break_LineWide" Tag should MOVE a 16 unless*:
   // *  If this workcenter is tied to the main line, and there is already a workcenter with a workstaiton where "Break_LineWide MOVEs a 16 in, even the first workstation in this workcenter can be 0  *
   // All other workstations within workcenter, "Break_LineWide" Tag should MOVE a 0 (not 16)
   63: [XIO(Break_1stStation) MOV(LN02_Main_Messages[90],LN02WGS01) ,XIC(Break_1stStation) MOV(LN02_1st_Station_Break_Code,LN02WGS01) ];
   64: [XIO(Break_1stStation) MOV(LN02_Main_Messages[91],LN02WGS02) ,XIC(Break_1stStation) MOV(0,LN02WGS02) ];
   65: [XIO(Break_1stStation) MOV(LN02_Main_Messages[92],LN02WGS03) ,XIC(Break_1stStation) MOV(0,LN02WGS03) ];
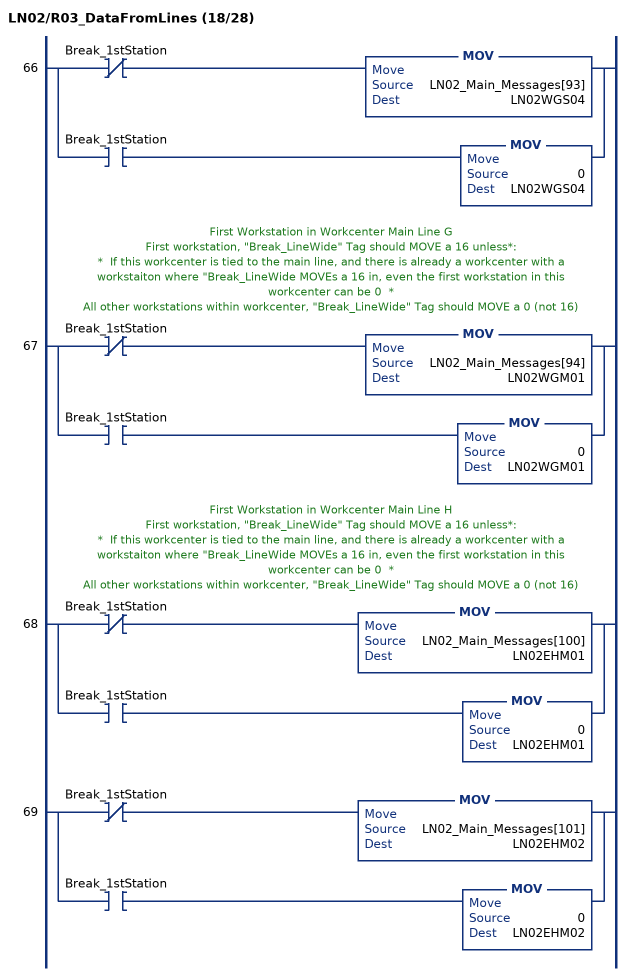
   66: [XIO(Break_1stStation) MOV(LN02_Main_Messages[93],LN02WGS04) ,XIC(Break_1stStation) MOV(0,LN02WGS04) ];
   // First Workstation in Workcenter Main Line G
   // First workstation, "Break_LineWide" Tag should MOVE a 16 unless*:
   // *  If this workcenter is tied to the main line, and there is already a workcenter with a workstaiton where "Break_LineWide MOVEs a 16 in, even the first workstation in this workcenter can be 0  *
   // All other workstations within workcenter, "Break_LineWide" Tag should MOVE a 0 (not 16)
   67: [XIO(Break_1stStation) MOV(LN02_Main_Messages[94],LN02WGM01) ,XIC(Break_1stStation) MOV(0,LN02WGM01) ];
   // First Workstation in Workcenter Main Line H
   // First workstation, "Break_LineWide" Tag should MOVE a 16 unless*:
   // *  If this workcenter is tied to the main line, and there is already a workcenter with a workstaiton where "Break_LineWide MOVEs a 16 in, even the first workstation in this workcenter can be 0  *
   // All other workstations within workcenter, "Break_LineWide" Tag should MOVE a 0 (not 16)
   68: [XIO(Break_1stStation) MOV(LN02_Main_Messages[100],LN02EHM01) ,XIC(Break_1stStation) MOV(0,LN02EHM01) ];
   69: [XIO(Break_1stStation) MOV(LN02_Main_Messages[101],LN02EHM02) ,XIC(Break_1stStation) MOV(0,LN02EHM02) ];
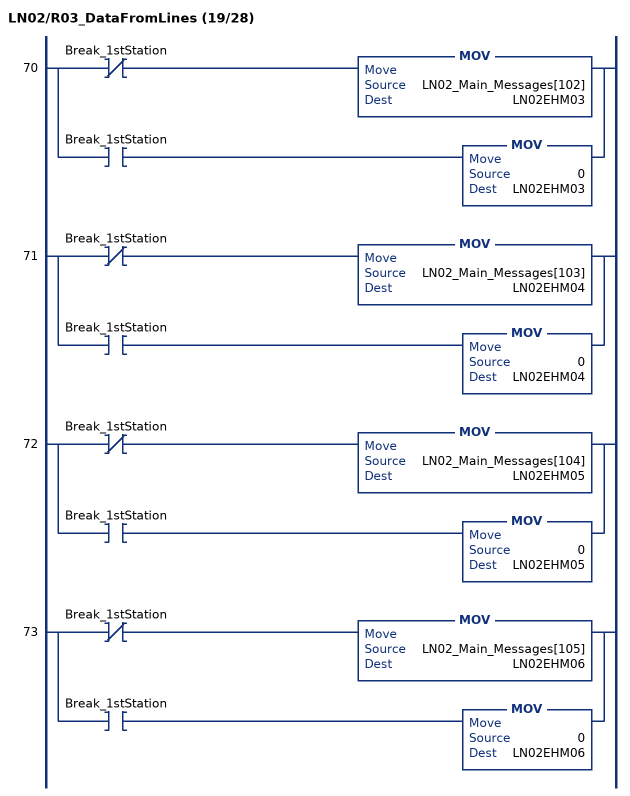
   70: [XIO(Break_1stStation) MOV(LN02_Main_Messages[102],LN02EHM03) ,XIC(Break_1stStation) MOV(0,LN02EHM03) ];
   71: [XIO(Break_1stStation) MOV(LN02_Main_Messages[103],LN02EHM04) ,XIC(Break_1stStation) MOV(0,LN02EHM04) ];
   72: [XIO(Break_1stStation) MOV(LN02_Main_Messages[104],LN02EHM05) ,XIC(Break_1stStation) MOV(0,LN02EHM05) ];
   73: [XIO(Break_1stStation) MOV(LN02_Main_Messages[105],LN02EHM06) ,XIC(Break_1stStation) MOV(0,LN02EHM06) ];
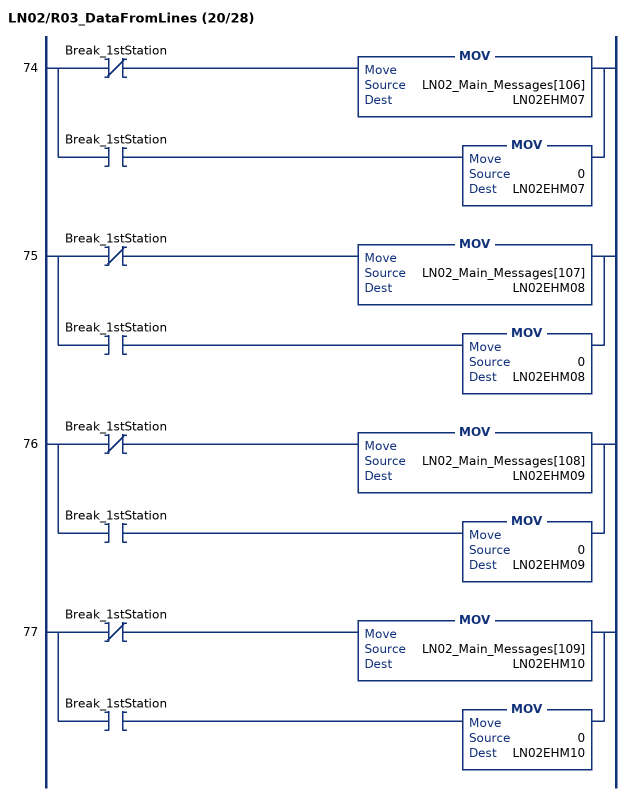
   74: [XIO(Break_1stStation) MOV(LN02_Main_Messages[106],LN02EHM07) ,XIC(Break_1stStation) MOV(0,LN02EHM07) ];
   75: [XIO(Break_1stStation) MOV(LN02_Main_Messages[107],LN02EHM08) ,XIC(Break_1stStation) MOV(0,LN02EHM08) ];
   76: [XIO(Break_1stStation) MOV(LN02_Main_Messages[108],LN02EHM09) ,XIC(Break_1stStation) MOV(0,LN02EHM09) ];
   77: [XIO(Break_1stStation) MOV(LN02_Main_Messages[109],LN02EHM10) ,XIC(Break_1stStation) MOV(0,LN02EHM10) ];
